% RSLogix 500 project BLUE_BANNER_HPW_SOME_TAGS_JULY_15_2021.RSS, saved by version 11.00.00.00 %
PROJECT "UNTITLED"    % processor: MicroLogix 1000 %

PROGRAM FILES
  LAD 2 "MAIN_PROG"  19 rungs
  LAD 3 "USER_FAULT"  18 rungs
  LAD 4 "HSC_INT"  5 rungs
  LAD 5 "STI_INT"  1 rungs
  LAD 6, 7, 8, 9, 10, 11, 12, 13, 14, 15, 16: only END

DATA FILES
  O0 OUTPUT  1 elements
  I1 INPUT  2 elements
  S2 STATUS  33 elements
  B3 BINARY  32 elements
  T4 TIMER  40 elements
  C5 COUNTER  32 elements
  R6 CONTROL  16 elements
  N7 INTEGER  105 elements

LADDER 2 "MAIN_PROG"
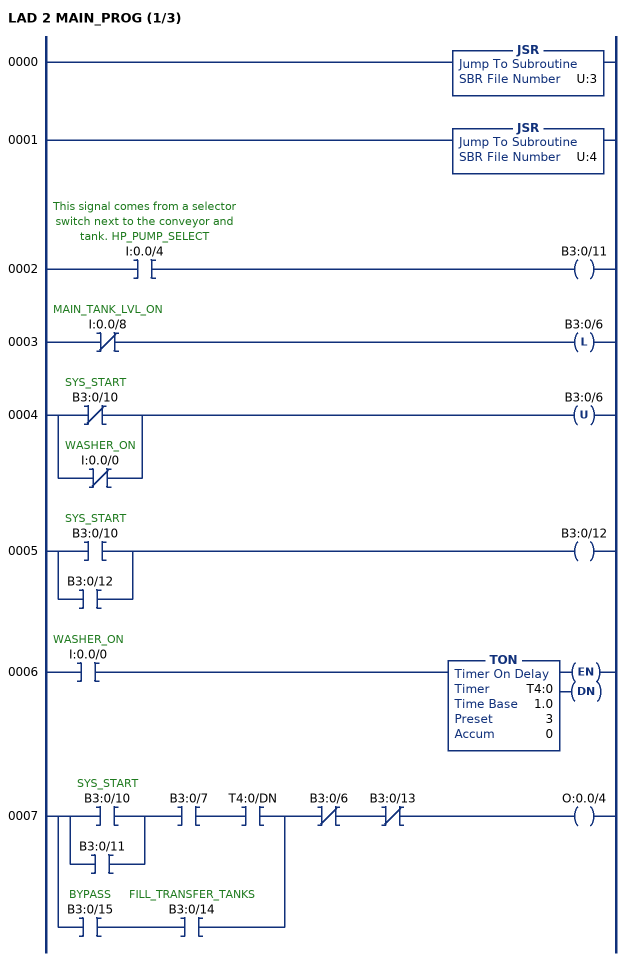
% Rung: 0 %
SOR JSR U:3 EOR
% Rung: 1 %
SOR JSR U:4 EOR
% Rung: 2 %
SOR XIC I:0.0/4 OTE B3:0/11 EOR
%   I:0.0/4  HP_PUMP_SELECT  "This signal comes from a selector switch next to the conveyor and tank." %
% Rung: 3 %
SOR XIO I:0.0/8 OTL B3:0/6 EOR
%   I:0.0/8  MAIN_TANK_LVL_ON %
% Rung: 4 %
SOR BST XIO B3:0/10 NXB XIO I:0.0/0 BND OTU B3:0/6 EOR
%   B3:0/10  SYS_START %
%   I:0.0/0  WASHER_ON %
% Rung: 5 %
SOR BST XIC B3:0/10 NXB XIC B3:0/12 BND OTE B3:0/12 EOR
%   B3:0/10  SYS_START %
% Rung: 6 %
SOR XIC I:0.0/0 TON T4:0 1.0 3 0 EOR
%   I:0.0/0  WASHER_ON %
% Rung: 7 %
SOR BST BST XIC B3:0/10 NXB XIC B3:0/11 BND XIC B3:0/7 XIC T4:0/DN NXB XIC B3:0/15 XIC B3:0/14 BND XIO B3:0/6 XIO B3:0/13 OTE O:0.0/4 EOR
%   B3:0/10  SYS_START %
%   B3:0/15  BYPASS %
%   B3:0/14  FILL_TRANSFER_TANKS %

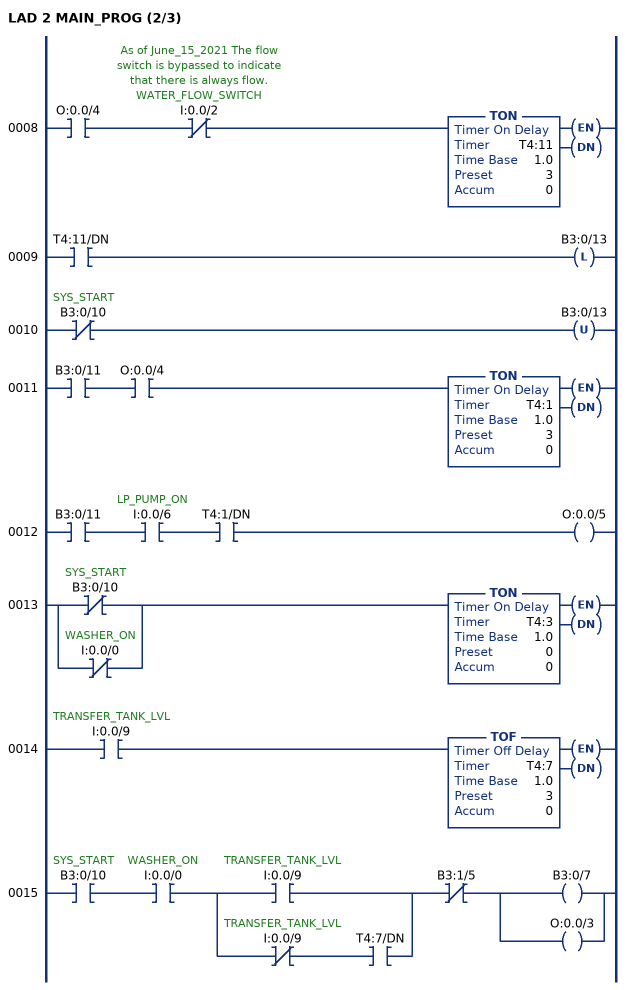
% Rung: 8 %
SOR XIC O:0.0/4 XIO I:0.0/2 TON T4:11 1.0 3 0 EOR
%   I:0.0/2  WATER_FLOW_SWITCH  "As of June_15_2021 The flow switch is bypassed to indicate that there is always flow." %
% Rung: 9 %
SOR XIC T4:11/DN OTL B3:0/13 EOR
% Rung: 10 %
SOR XIO B3:0/10 OTU B3:0/13 EOR
%   B3:0/10  SYS_START %
% Rung: 11 %
SOR XIC B3:0/11 XIC O:0.0/4 TON T4:1 1.0 3 0 EOR
% Rung: 12 %
SOR XIC B3:0/11 XIC I:0.0/6 XIC T4:1/DN OTE O:0.0/5 EOR
%   I:0.0/6  LP_PUMP_ON %
% Rung: 13 %
SOR BST XIO B3:0/10 NXB XIO I:0.0/0 BND TON T4:3 1.0 0 0 EOR
%   B3:0/10  SYS_START %
%   I:0.0/0  WASHER_ON %
% Rung: 14 %
SOR XIC I:0.0/9 TOF T4:7 1.0 3 0 EOR
%   I:0.0/9  TRANSFER_TANK_LVL %
% Rung: 15 %
SOR XIC B3:0/10 XIC I:0.0/0 BST XIC I:0.0/9 NXB XIO I:0.0/9 XIC T4:7/DN BND XIO B3:1/5 BST OTE B3:0/7 NXB OTE O:0.0/3 BND EOR
%   B3:0/10  SYS_START %
%   I:0.0/0  WASHER_ON %
%   I:0.0/9  TRANSFER_TANK_LVL %

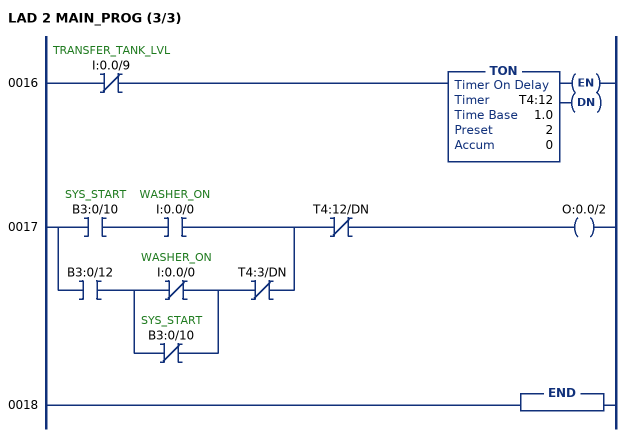
% Rung: 16 %
SOR XIO I:0.0/9 TON T4:12 1.0 2 0 EOR
%   I:0.0/9  TRANSFER_TANK_LVL %
% Rung: 17 %
SOR BST XIC B3:0/10 XIC I:0.0/0 NXB XIC B3:0/12 BST XIO I:0.0/0 NXB XIO B3:0/10 BND XIO T4:3/DN BND XIO T4:12/DN OTE O:0.0/2 EOR
%   B3:0/10  SYS_START %
%   I:0.0/0  WASHER_ON %
% Rung: 18 %
SOR END EOR

LADDER 3 "USER_FAULT"
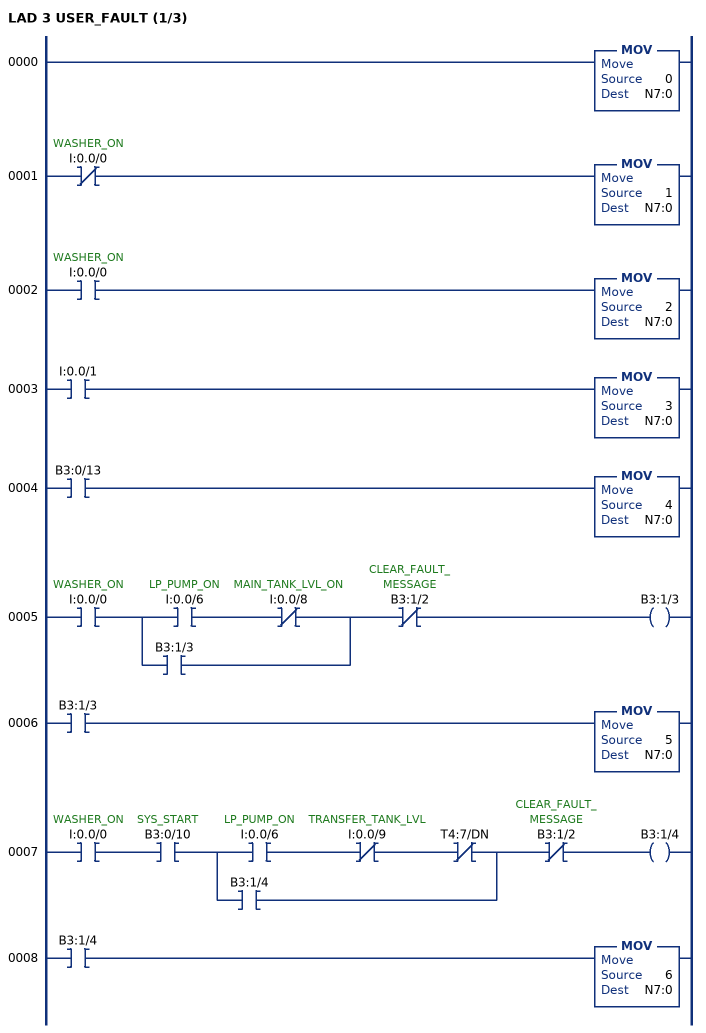
% Rung: 0 %
SOR MOV 0 N7:0 EOR
% Rung: 1 %
SOR XIO I:0.0/0 MOV 1 N7:0 EOR
%   I:0.0/0  WASHER_ON %
% Rung: 2 %
SOR XIC I:0.0/0 MOV 2 N7:0 EOR
%   I:0.0/0  WASHER_ON %
% Rung: 3 %
SOR XIC I:0.0/1 MOV 3 N7:0 EOR
% Rung: 4 %
SOR XIC B3:0/13 MOV 4 N7:0 EOR
% Rung: 5 %
SOR XIC I:0.0/0 BST XIC I:0.0/6 XIO I:0.0/8 NXB XIC B3:1/3 BND XIO B3:1/2 OTE B3:1/3 EOR
%   I:0.0/0  WASHER_ON %
%   I:0.0/6  LP_PUMP_ON %
%   I:0.0/8  MAIN_TANK_LVL_ON %
%   B3:1/2  CLEAR_FAULT_MESSAGE %
% Rung: 6 %
SOR XIC B3:1/3 MOV 5 N7:0 EOR
% Rung: 7 %
SOR XIC I:0.0/0 XIC B3:0/10 BST XIC I:0.0/6 XIO I:0.0/9 XIO T4:7/DN NXB XIC B3:1/4 BND XIO B3:1/2 OTE B3:1/4 EOR
%   I:0.0/0  WASHER_ON %
%   B3:0/10  SYS_START %
%   I:0.0/6  LP_PUMP_ON %
%   I:0.0/9  TRANSFER_TANK_LVL %
%   B3:1/2  CLEAR_FAULT_MESSAGE %
% Rung: 8 %
SOR XIC B3:1/4 MOV 6 N7:0 EOR

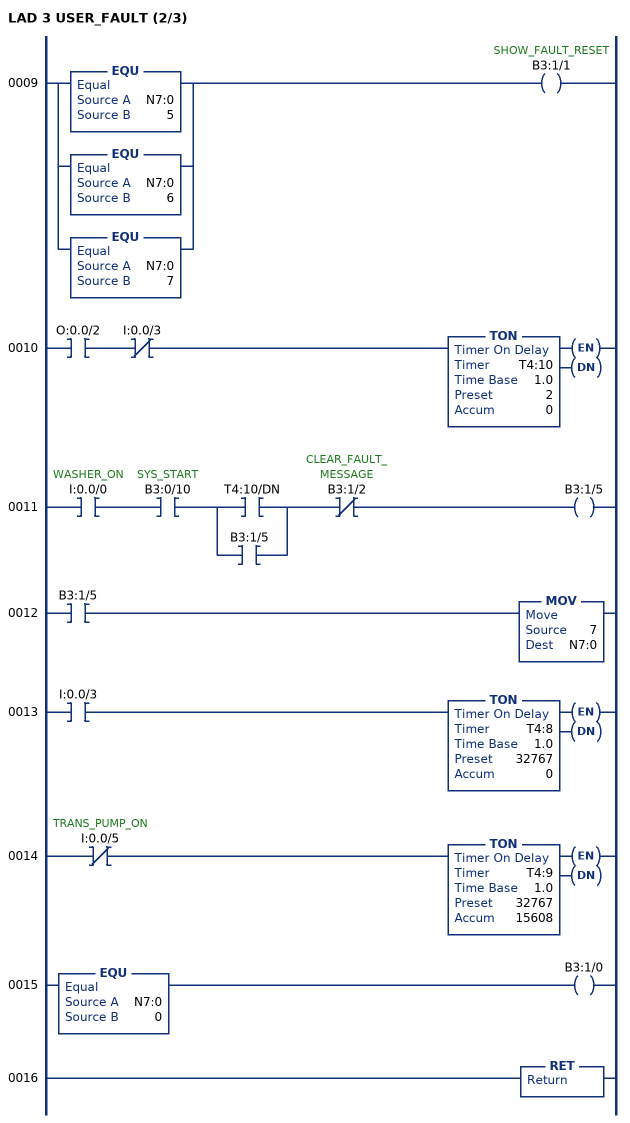
% Rung: 9 %
SOR BST BST EQU N7:0 5 NXB EQU N7:0 6 BND NXB EQU N7:0 7 BND OTE B3:1/1 EOR
%   B3:1/1  SHOW_FAULT_RESET %
% Rung: 10 %
SOR XIC O:0.0/2 XIO I:0.0/3 TON T4:10 1.0 2 0 EOR
% Rung: 11 %
SOR XIC I:0.0/0 XIC B3:0/10 BST XIC T4:10/DN NXB XIC B3:1/5 BND XIO B3:1/2 OTE B3:1/5 EOR
%   I:0.0/0  WASHER_ON %
%   B3:0/10  SYS_START %
%   B3:1/2  CLEAR_FAULT_MESSAGE %
% Rung: 12 %
SOR XIC B3:1/5 MOV 7 N7:0 EOR
% Rung: 13 %
SOR XIC I:0.0/3 TON T4:8 1.0 32767 0 EOR
% Rung: 14 %
SOR XIO I:0.0/5 TON T4:9 1.0 32767 15608 EOR
%   I:0.0/5  TRANS_PUMP_ON %
% Rung: 15 %
SOR EQU N7:0 0 OTE B3:1/0 EOR
% Rung: 16 %
SOR RET EOR

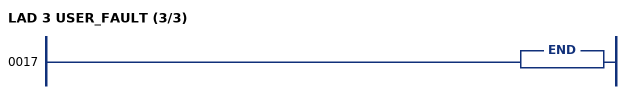
% Rung: 17 %
SOR END EOR

LADDER 4 "HSC_INT"
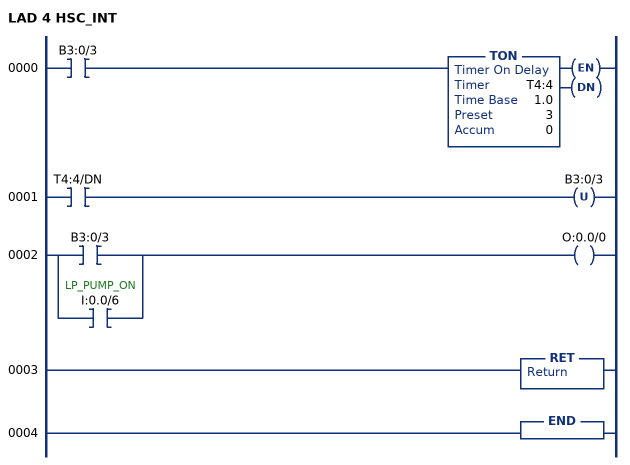
% Rung: 0 %
SOR XIC B3:0/3 TON T4:4 1.0 3 0 EOR
% Rung: 1 %
SOR XIC T4:4/DN OTU B3:0/3 EOR
% Rung: 2 %
SOR BST XIC B3:0/3 NXB XIC I:0.0/6 BND OTE O:0.0/0 EOR
%   I:0.0/6  LP_PUMP_ON %
% Rung: 3 %
SOR RET EOR
% Rung: 4 %
SOR END EOR

OTHER DOCUMENTED ADDRESSES
  I:0.0/7  HP_PUMP_ON
  T4:0.PRE  START_DELAY
  T4:1.PRE  HP_START_DELAY
  T4:3.PRE  TRANS_OFF_DELAY
  T4:4.PRE  PRIME_DUR
  T4:7.PRE  TRANS_TANK_LOW_DELAY
  T4:8.ACC  TRANS_PUMP_RUN_TIME
  T4:9.ACC  TRANS_PUMP_OFF_TIME

DATA TABLE (non-zero values as saved)
DATA B3
% B3:0 % 0X9400 0X0000 0X0000 0X0000 0X0000 0X0000 0X0000 0X0000 0X0000 0X0000
DATA T4
% .PRE .ACC %
% T4:0 % 3 0
% T4:1 % 3 0
% T4:2 % 2 0
% T4:4 % 3 0
% T4:5 % 10 0
% T4:6 % 50 0
% T4:7 % 3 0
% T4:8 % 32767 0
% T4:9 % 32767 15608
% T4:10 % 2 0
% T4:11 % 3 0
% T4:12 % 2 0
DATA N7
% N7:0 % 1 0 0 0 0 0 0 0 0 0
